(*
An interface that represents an object callable through various systems. 
*)
INTERFACE I_Callable EXTENDS I_Debug

(*
This method provides a standardized way for other objects to interact with the object that owns it.
*)
METHOD Call
VAR_INPUT
	iArg		: I_Arg;
END_VAR
END_METHOD

END_INTERFACE

(* stored: Version 1.1.0.1
   Itf I_Callable: Id {50cf3f2b-50a0-4a04-bbe5-39ba2a7999af}
   Method Call: Id {c7d88913-b4b8-4b49-bfda-281bb631abd0} *)
